DATA_BLOCK "DB_LSZ_Type"
TITLE =%version: 0.06 % CN: 20
//History:
//This version  %created_by: nlhdl %
//              %date_created: maandag 6 juli 2015 10:23:21 %
//              %release: VI_CONV/RA_Dev_Oakham %
//
//Modification History:                                   By:    Date:     Rev:
//----------------------------------------------------  -------  --------  -----
//7324: ECS-P General from the RD to RA for platform    nlHdL    06-07-15   0.06
//15797: Keyword release added                          nlwwij   26-09-13   0.06
//PR6725 Remove report Offline when Status 1 is true    nlple    12-04-11   0.05
//CR6389 Changed statusses and OS/GS                    nlJBax   14-01-11   0.04
//CR5764 Status UDT Update name change                  nlHdL    05-10-10   0.03
//CR5712 Not used errors have number -1                 nlHdL    24-09-10   0.02
//Initial Revision                                      inpna    17-09-10   0.01
//
FAMILY : General
VERSION : 0.0


  STRUCT
   Type_Component : BYTE ;	//Type of the component (1 = Section, 0 = Other)
   Record_Length : BYTE  := B#16#16;	//Number of the Detailed Status in the UDT
   Status : ARRAY  [1 .. 16 ] OF "UDT_Comp_Status";
  END_STRUCT ;
BEGIN
   Type_Component := B#16#0;
   Record_Length := B#16#16;
   Status[1].HMI_Text_Number := -1;
   Status[1].Overall_Status_Relation := B#16#0;
   Status[1].General_Status_Relation := B#16#0;
   Status[2].HMI_Text_Number := -1;
   Status[2].Overall_Status_Relation := B#16#0;
   Status[2].General_Status_Relation := B#16#0;
   Status[3].HMI_Text_Number := -1;
   Status[3].Overall_Status_Relation := B#16#0;
   Status[3].General_Status_Relation := B#16#0;
   Status[4].HMI_Text_Number := -1;
   Status[4].Overall_Status_Relation := B#16#0;
   Status[4].General_Status_Relation := B#16#0;
   Status[5].HMI_Text_Number := -1;
   Status[5].Overall_Status_Relation := B#16#0;
   Status[5].General_Status_Relation := B#16#0;
   Status[6].HMI_Text_Number := -1;
   Status[6].Overall_Status_Relation := B#16#0;
   Status[6].General_Status_Relation := B#16#0;
   Status[7].HMI_Text_Number := -1;
   Status[7].Overall_Status_Relation := B#16#0;
   Status[7].General_Status_Relation := B#16#0;
   Status[8].HMI_Text_Number := -1;
   Status[8].Overall_Status_Relation := B#16#0;
   Status[8].General_Status_Relation := B#16#0;
   Status[9].HMI_Text_Number := -1;
   Status[9].Overall_Status_Relation := B#16#0;
   Status[9].General_Status_Relation := B#16#0;
   Status[10].HMI_Text_Number := -1;
   Status[10].Overall_Status_Relation := B#16#0;
   Status[10].General_Status_Relation := B#16#0;
   Status[11].HMI_Text_Number := -1;
   Status[11].Overall_Status_Relation := B#16#0;
   Status[11].General_Status_Relation := B#16#0;
   Status[12].HMI_Text_Number := -1;
   Status[12].Overall_Status_Relation := B#16#0;
   Status[12].General_Status_Relation := B#16#0;
   Status[13].HMI_Text_Number := -1;
   Status[13].Overall_Status_Relation := B#16#0;
   Status[13].General_Status_Relation := B#16#0;
   Status[14].HMI_Text_Number := -1;
   Status[14].Overall_Status_Relation := B#16#0;
   Status[14].General_Status_Relation := B#16#0;
   Status[15].HMI_Text_Number := -1;
   Status[15].Overall_Status_Relation := B#16#0;
   Status[15].General_Status_Relation := B#16#0;
   Status[16].HMI_Text_Number := -1;
   Status[16].Overall_Status_Relation := B#16#0;
   Status[16].General_Status_Relation := B#16#0;
END_DATA_BLOCK

